FUNCTION_BLOCK ObserveCrane EXTENDS HardwareObservationBase
VAR_INPUT
END_VAR
VAR_OUTPUT
END_VAR
VAR
	m_ptrCrane: POINTER TO Crane;
	m_ptrCraneWP: POINTER TO xPPUProduct;
	
	m_rtAtStack: R_TRIG;
	m_rtAtLSC: R_TRIG;
	m_rtAtStamp: R_TRIG;
	
	m_resetCranePos: BOOL;
END_VAR

METHOD FB_init : BOOL
VAR_INPUT
	bInitRetains : BOOL; // if TRUE, the retain variables are initialized (warm start / cold start)
	bInCopyCode : BOOL;  // if TRUE, the instance afterwards gets moved into the copy code (online change)

	i_ptrCrane: POINTER TO Crane;
	i_ptrWP: POINTER TO IProduct;
END_VAR
m_ptrCrane := i_ptrCrane;
IF NOT __QUERYPOINTER(i_ptrWP^, m_ptrCraneWP) THEN
	FB_init := FALSE;
END_IF
END_METHOD

METHOD  ResetDefinition : BOOL
VAR_INPUT
END_VAR
m_resetCranePos := TRUE;
END_METHOD

(* Update an instance of ProcessState with the part of the process that can be observed by this Hardware Interface. *)
METHOD UpdateProcessObservation : BOOL
VAR_IN_OUT
	io_processState: ProcessState;
END_VAR
io_processState.UpdateState_Binary(EProcessVariables.Crane_AtStack, m_ptrCrane^.AtStack, i_force := TRUE);
io_processState.UpdateState_Binary(EProcessVariables.Crane_AtStamp, m_ptrCrane^.AtStamp, i_force := TRUE);
io_processState.UpdateState_Binary(EProcessVariables.Crane_AtLSC, m_ptrCrane^.AtConveyor, i_force := TRUE);
io_processState.UpdateState_Binary(EProcessVariables.Crane_HoldingWorkpiece, m_ptrCrane^.o_VacuumGripper.WPTaken, i_force := TRUE);
io_processState.UpdateState_Binary(EProcessVariables.Crane_CylinderExtended, m_ptrCrane^.o_MonostableCylinder.Extended, i_force := TRUE);
io_processState.UpdateState_Binary(EProcessVariables.Crane_CylinderRetracted, m_ptrCrane^.o_MonostableCylinder.Retracted, i_force := TRUE);
io_processState.UpdateState_Numeric(EProcessVariables.Crane_Angle, INT_TO_LREAL(m_ptrCrane^.o_Angle), i_force := TRUE);

m_rtAtStack(CLK := m_ptrCrane^.AtStack);
m_rtAtStamp(CLK := m_ptrCrane^.AtStamp);
m_rtAtLSC(CLK := m_ptrCrane^.AtConveyor);

IF m_rtAtStack.Q OR m_rtAtStamp.Q OR m_rtAtLSC.Q THEN
	io_processState.UpdateState_Defined(EProcessVariables.Crane_AtStack, TRUE);
	io_processState.UpdateState_Defined(EProcessVariables.Crane_AtStamp, TRUE);
	io_processState.UpdateState_Defined(EProcessVariables.Crane_AtLSC, TRUE);
	io_processState.UpdateState_Defined(EProcessVariables.Crane_Angle, TRUE);	
END_IF
IF m_resetCranePos THEN
	io_processState.UpdateState_Defined(EProcessVariables.Crane_AtStack, FALSE);
	io_processState.UpdateState_Defined(EProcessVariables.Crane_AtStamp, FALSE);
	io_processState.UpdateState_Defined(EProcessVariables.Crane_AtLSC, FALSE);
	io_processState.UpdateState_Defined(EProcessVariables.Crane_Angle, FALSE);
	
	m_resetCranePos := FALSE;
END_IF

io_processState.UpdateState_Defined(EProcessVariables.Crane_HoldingWorkpiece, TRUE);
io_processState.UpdateState_Defined(EProcessVariables.Crane_CylinderExtended, TRUE);
io_processState.UpdateState_Defined(EProcessVariables.Crane_CylinderRetracted, TRUE);



// update WP info (if there are sensors available), then update the process variables list
io_processState.UpdateState_Numeric(EProcessVariables.Crane_ProductType, UINT_TO_LREAL(m_ptrCraneWP^.Material), TRUE);
io_processState.UpdateState_Defined(EProcessVariables.Crane_ProductType, TRUE);
END_METHOD

END_FUNCTION_BLOCK

(* stored: Version 1.1.0.1, ProductVersion 3.1.4024.12
   POU ObserveCrane: Id {4954d856-72f9-465f-a8a6-2f8aa4b61f6c}, SpecialFunc None
   Method FB_init: Id {70e3b3ab-124c-45c5-a113-c1f4961d83e3}
   Method ResetDefinition: Id {1b1f8bfe-8e46-475f-9b81-d1e60cd83af8}
   Method UpdateProcessObservation: Id {e8ee6704-ca71-439d-9fa8-f0ee43b90df7} *)
